Omron CX-Programmer project NewProject (CX-Programmer 9.63)

# PLC NewPLC1: CJ2M CPU11

## Global symbols (name address type ; comment)
0.00 BOOL  ; Button
100.02 BOOL  ; InPosition
1.00 BOOL  ; CravamentoOK_C1
1.01 BOOL  ; CravamentoOK_C2
W0.00 BOOL  ; CravamentoOK_C1
W0.01 BOOL  ; CravamentoOK_C2
W0.02 BOOL  ; Sinal_Start
W0.03 BOOL  ; Sinal_STOP
W0.04 BOOL  ; ResultOK_Inspection
W0.05 BOOL  ; ResultNOK_Inspection
W0.06 BOOL  ; Emergência
Eixo_Y Eixo_Y
eixo_Y Eixo_Y

## Program CravamentoSolas (cyclic task 0)
Local symbols
Emergência 1.07 BOOL  ; aux
ResultNOK 1.05 BOOL
ResultOK 1.04 BOOL
Sinal_NOK 1.03 BOOL
Sinal_START 1.02 BOOL
Sinal_STOP 1.03 BOOL
inPos 1.07 BOOL
w BOOL
ww0 UINT

### Section Saidas

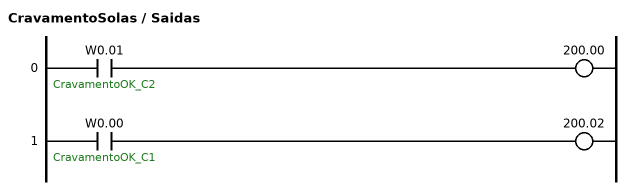
; rung 0
LD W0.01  ; CravamentoOK_C2
OUT 200.00
; rung 1
LD W0.00  ; CravamentoOK_C1
OUT 200.02

### Section Entradas

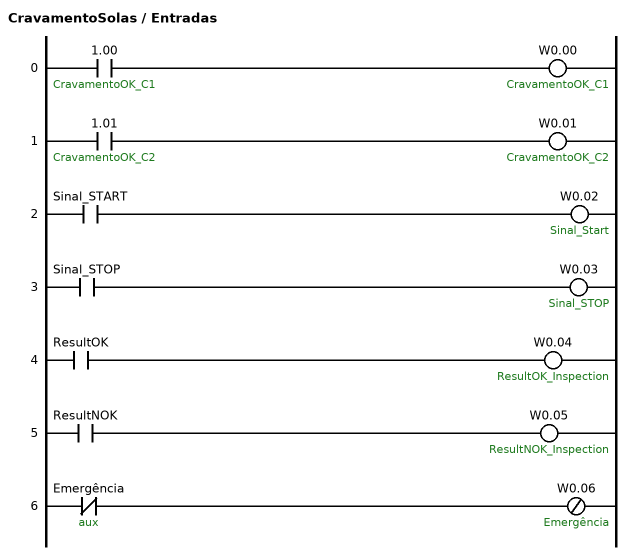
; rung 0
LD 1.00  ; CravamentoOK_C1
OUT W0.00  ; CravamentoOK_C1
; rung 1
LD 1.01  ; CravamentoOK_C2
OUT W0.01  ; CravamentoOK_C2
; rung 2
LD Sinal_START
OUT W0.02  ; Sinal_Start
; rung 3
LD Sinal_STOP
OUT W0.03  ; Sinal_STOP
; rung 4
LD ResultOK
OUT W0.04  ; ResultOK_Inspection
; rung 5
LD ResultNOK
OUT W0.05  ; ResultNOK_Inspection
; rung 6
LDNOT Emergência  ; aux
OUTNOT W0.06  ; Emergência

### Section ModoManual

### Section ModoAutomatico

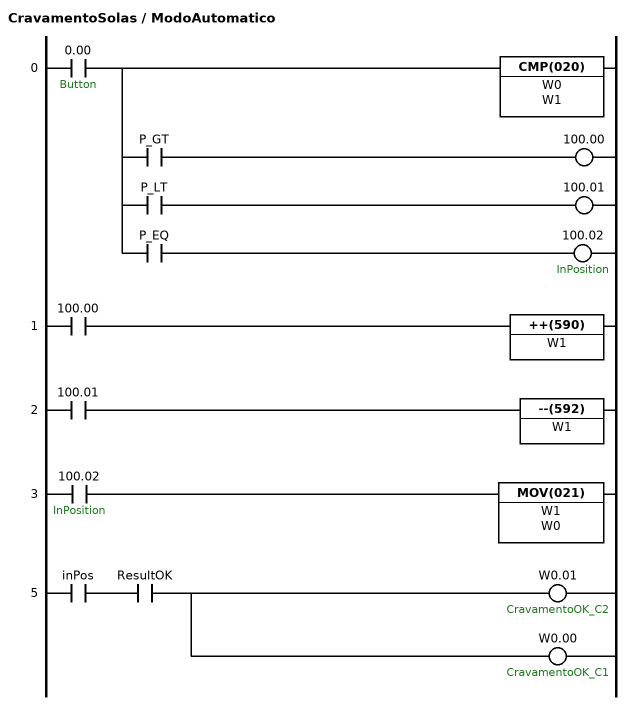
; rung 0
LD 0.00  ; Button
OUT TR0
CMP(020) W0 W1
AND P_GT
OUT 100.00
LD TR0
AND P_LT
OUT 100.01
LD TR0
AND P_EQ
OUT 100.02  ; InPosition
; rung 1
LD 100.00
++(590) W1
; rung 2
LD 100.01
--(592) W1
; rung 3
LD 100.02  ; InPosition
MOV(021) W1 W0
; rung 4
; cells of this rung as drawn
  row 1 col 0: LD Sinal_START
  row 1 col 1: CALL Eixo_Y : Eixo_Y ()
  row 1 col 3: wire
  row 1 col 4: wire
  row 1 col 5: wire
  row 1 col 6: OUT ResultOK
  row 2 col 3: wire
  row 2 col 4: wire
  row 2 col 5: wire
  row 2 col 6: OUT inPos
  vertical links (row, left of col): 
; rung 5
LD inPos
AND ResultOK
OUT W0.01  ; CravamentoOK_C2
OUT W0.00  ; CravamentoOK_C1

### Section Alarmes

### Section Manutencao

### Section END
; rung 0
END(001)

## Function block Eixo_Y
VAR_INPUT
  MovePos : INT;
  CurPos : INT;
END_VAR
VAR_OUTPUT
  InPosition : INT;
END_VAR

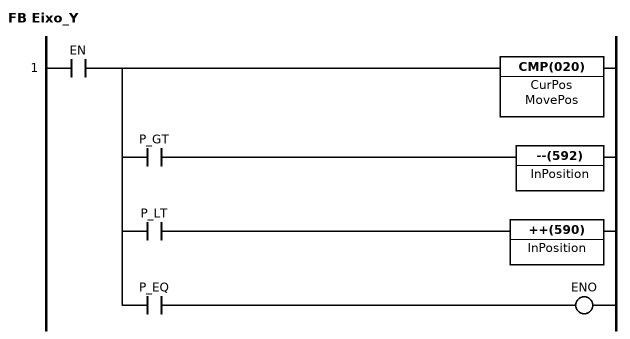
; rung 1
LD EN
OUT TR0
CMP(020) CurPos MovePos
AND P_GT
--(592) InPosition
LD TR0
AND P_LT
++(590) InPosition
LD TR0
AND P_EQ
OUT ENO